FUNCTION F_RAW_TO_PHYS (* Convert ISOBUS raw UDINT to physical REAL value. ISOBUS formula: display = (raw + offset) * scale Example: raw=50000, scale=0.01, offset=-100000 DINT(50000) + (-100000) = -50000 REAL(-50000) 0.01     = -500.0 *)
  (* Standard: 61499-2; Description: Copyright (c) 2026 Meisterschulen am Ostbahnhof This program and the accompanying materials are made available under the terms of the Eclipse Public License 2.0 which is available at https://www.eclipse.org/legal/epl-2.0/ SPDX-License-Identifier: EPL-2.0 *)
  (* Version 1.0, 2026-04-14, Franz Höpfinger, Meisterschulen am Ostbahnhof *)
  PACKAGE isobus::UT::io::NumericValue;
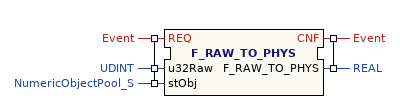
  EVENT_INPUT
    REQ WITH u32Raw, stObj;
  END_EVENT
  EVENT_OUTPUT
    CNF WITH F_RAW_TO_PHYS;
  END_EVENT
  VAR_INPUT
    u32Raw : UDINT;
    stObj : isobus::UT::io::NumericValue::NumericObjectPool_S;
  END_VAR
  VAR_OUTPUT
    F_RAW_TO_PHYS : REAL;
  END_VAR
  BODY IN ST:
PACKAGE isobus::UT::io::NumericValue;

(* Convert ISOBUS raw UDINT to physical REAL value.
 * ISOBUS formula: display = (raw + offset) * scale
 *
 * Example: raw=50000, scale=0.01, offset=-100000 DINT(50000) + (-100000) = -50000 REAL(-50000) *
 * 0.01     = -500.0 *)
FUNCTION F_RAW_TO_PHYS : REAL

VAR_INPUT
	u32Raw : UDINT;
	stObj : NumericObjectPool_S;
END_VAR

F_RAW_TO_PHYS := DINT_TO_REAL(UDINT_TO_DINT(u32Raw) + stObj.i32Offset) * stObj.r32Scale;

END_FUNCTION
  END_BODY
END_FUNCTION
